{attribute 'hide'}
FUNCTION_BLOCK FB_Test_Base EXTENDS FB_TestBase

(******************************************************************************
Baustein: FB_Test_Base.cleanup
Spezifikation: doc/Spezifikation.pdf, Kap. x.y.z
-------------------------------------------------------------------------------
erstellt:
von:
Geändert:
von:
-------------------------------------------------------------------------------
Beschreibung
Diese Methode...

-------------------------------------------------------------------------------
Input
-

Output
-
******************************************************************************)
METHOD PUBLIC cleanup : ERetCode_t
VAR_INPUT
END_VAR

	cleanup := ERetCode_t.eRetDone;
END_METHOD

(******************************************************************************
Baustein: FB_Test_Base.execute
Spezifikation: doc/Spezifikation.pdf, Kap. x.y.z
-------------------------------------------------------------------------------
erstellt:
von:
Geändert:
von:
-------------------------------------------------------------------------------
Beschreibung
Diese Methode...

-------------------------------------------------------------------------------
Input
-

Output
-
******************************************************************************)
METHOD PUBLIC execute : ERetCode_t
VAR_INPUT
END_VAR
VAR
	bValue1   : ARRAY[0..10] OF BOOL;
	bValue2   : ARRAY[0..10] OF BOOL;
	s8Value1  : ARRAY[0..10] OF SINT;
	s8Value2  : ARRAY[0..10] OF SINT;
	u8Value1  : ARRAY[0..10] OF USINT;
	u8Value2  : ARRAY[0..10] OF USINT;	
	s16Value1 : ARRAY[0..10] OF INT;
	s16Value2 : ARRAY[0..10] OF INT;
	u16Value1 : ARRAY[0..10] OF UINT;
	u16Value2 : ARRAY[0..10] OF UINT;		
	s32Value1 : ARRAY[0..10] OF DINT;
	s32Value2 : ARRAY[0..10] OF DINT;
	u32Value1 : ARRAY[0..10] OF UDINT;
	u32Value2 : ARRAY[0..10] OF UDINT;	
	r32Value1 : ARRAY[0..10] OF REAL;
	r32Value2 : ARRAY[0..10] OF REAL;
	r64Value1 : ARRAY[0..10] OF LREAL;
	r64Value2 : ARRAY[0..10] OF LREAL;
	strValue1 : ARRAY[0..10] OF STRING;
	strValue2 : ARRAY[0..10] OF STRING;
END_VAR


	bValue1[0] := TRUE;
	bValue2[0] := TRUE;
	
	setMessage('Teste Datentyp BOOL');
	assert.EQUAL(bValue1[0], bValue2[0]);
	
	setMessage('Teste Datentyp Array of BOOL');
	assert.EQUAL(bValue1, bValue2);

(**********************************************) 
	
	s8Value1[0] := 32;
	s8Value2[0] := 32;
	
	setMessage('Teste Datentyp SINT');
	assert.EQUAL(s8Value1[0], s8Value2[0]);

	setMessage('Teste Datentyp Array of SINT');
	assert.EQUAL(s8Value1, s8Value2);
(**********************************************) 	

	u8Value1[0] := 34;
	u8Value2[0] := 34;
	
	setMessage('Teste Datentyp USINT');
	assert.EQUAL(u8Value1[0], u8Value2[0]);

	setMessage('Teste Datentyp Array of USINT');
	assert.EQUAL(u8Value1, u8Value2);
(**********************************************) 	
	
	s16Value1[0] := 1323;
	s16Value2[0] := 1323;
	
	setMessage('Teste Datentyp INT');
	assert.EQUAL(s16Value1[0], s16Value2[0]);

	setMessage('Teste Datentyp Array of INT');
	assert.EQUAL(s16Value1, s16Value2);
(**********************************************) 	

	u16Value1[0] := 3124;
	u16Value2[0] := 3124;
	
	setMessage('Teste Datentyp UINT');
	assert.EQUAL(u16Value1[0] , u16Value2[0] );

	setMessage('Teste Datentyp Array of UINT');
	assert.EQUAL(u16Value1 , u16Value2);
(**********************************************) 	

	s32Value1[0] := 1244;
	s32Value2[0] := 1244;
	
	setMessage('Teste Datentyp DINT');
	assert.EQUAL(s32Value1[0], s32Value2[0]);

	setMessage('Teste Datentyp Array of DINT');
	assert.EQUAL(s32Value1, s32Value2);
(**********************************************) 	

	u32Value1[0] := 4344;
	u32Value2[0] := 4344;
	
	setMessage('Teste Datentyp UDINT');
	assert.EQUAL(u32Value1[0], u32Value2[0]);

	setMessage('Teste Datentyp Array of UDINT');
	assert.EQUAL(u32Value1, u32Value2);
(**********************************************) 	

	r32Value1[0] := 133.53245;
	r32Value2[0] := 133.53245;
	
	setMessage('Teste Datentyp REAL');
	assert.EQUAL(r32Value1[0], r32Value2[0]);

	setMessage('Teste Datentyp Array of REAL');
	assert.EQUAL(r32Value1, r32Value2);
(**********************************************) 	

	r64Value1[0] := 1232.53325;
	r64Value2[0] := 1232.53325;

	setMessage('Teste Datentyp LREAL');
	assert.EQUAL(r64Value1[0], r64Value2[0]);

	setMessage('Teste Datentyp Array of LREAL');
	assert.EQUAL(r64Value1, r64Value2);

(**********************************************) 	

	strValue1[0] := 'Hallo Welt';
	strValue2[0] := 'Hallo Welt';

	setMessage('Teste Datentyp String ist gleich');
	assert.StringEqual(ADR(strValue1[0]), ADR(strValue2[0]));

	//setMessage('Teste Datentyp Array of String ist gleich');
	//assertEQUAL(strValue1, strValue2);

	strValue1[0] := 'Hallo Well';
	strValue2[0] := 'Hallo Welt';
	
	setMessage('Teste Datentyp String ist ungleich');
	assert.StringNotEqual(ADR(strValue1[0]), ADR(strValue2[0]));

	//setMessage('Teste Datentyp Array of String ist ungleich');
	//assert.NotEQUAL(strValue1, strValue2);
	
(**********************************************) 	





	execute := ERetCode_t.eRetDone;
END_METHOD

(******************************************************************************
Baustein: FB_Test_Base.prepare
Spezifikation: doc/Spezifikation.pdf, Kap. x.y.z
-------------------------------------------------------------------------------
erstellt:
von:
Geändert:
von:
-------------------------------------------------------------------------------
Beschreibung
Diese Methode...

-------------------------------------------------------------------------------
Input
-

Output
-
******************************************************************************)
METHOD PUBLIC prepare : ERetCode_t
VAR_INPUT
END_VAR

	prepare := ERetCode_t.eRetDone;
END_METHOD

END_FUNCTION_BLOCK

(* stored: Version 1.1.0.1, ProductVersion 3.1.4024.13
   POU FB_Test_Base: Id {f4823231-d10b-40e2-9073-1f2bc0a0599a}, SpecialFunc None
   Method cleanup: Id {49bced59-0780-425b-9290-17b9f069ca47}
   Method execute: Id {f50564e1-c200-4dfb-bffc-789888944368}
   Method prepare: Id {e23e127a-3b2e-47a3-9516-8405d2c66c55} *)
